// TIA Portal V18 export
// export: Created 2026-03-12T16:04:35.3703987Z, ExportSetting WithDefaults, DisplayName Totally Integrated Automation Portal, DisplayVersion V18 Update 5, DisplayName TIA Portal Openness, DisplayVersion V18 Update 5, DisplayName TIA Portal Version Control Interface, DisplayVersion V18, DisplayName SINAMICS Startdrive Advanced, DisplayVersion V18, DisplayName SINAMICS Startdrive G130, G150, S120, S150, SINAMICS MV, S210, DisplayVersion V18, DisplayName SINAMICS Startdrive G110M, G120, G120C, G120D, G120P, G115D, DisplayVersion V18, DisplayName STEP 7 Professional, DisplayVersion V18 Update 5, DisplayName STEP 7 Safety, DisplayVersion V18, DisplayName WinCC Professional, DisplayVersion V18 Update 5
FUNCTION_BLOCK "FB LIMITES_OPERACAO_SENSOR"   // FB25, LAD
{ S7_Optimized_Access := 'TRUE' }
VERSION : 0.1
// stored: AutoNumber true, IsIECCheckEnabled false, IsRetainMemResEnabled false, MemoryReserve 100, SetENOAutomatically false, UDAEnableTagReadback false
   VAR_INPUT
      STATUS_SENSOR : Real;
      COMANDO : Int;
      COMANDO_VALOR : Int;
      ENTRADA_VALOR_MUITO_BAIXO : Real;
      ENTRADA_VALOR_BAIXO : Real;
      ENTRADA_VALOR_ALTO : Real;
      ENTRADA_VALOR_MUITO_ALTO : Real;
      COMANDO_MANUTENCAO : Bool;
      SEM_SINAL_4mA : Bool;
   END_VAR
   VAR_OUTPUT
      SAIDA_LEITURA_MUITO_BAIXA : Bool;
      SAIDA_LEITURA_BAIXO : Bool;
      SAIDA_LEITURA_ALTO : Bool;
      SAIDA_LEITURA_MUITO_ALTO : Bool;
   END_VAR
   VAR_IN_OUT
      VALOR_MUITO_BAIXO : Real;
      VALOR_BAIXO : Real;
      VALOR_ALTO : Real;
      VALOR_MUITO_ALTO : Real;
   END_VAR
   VAR
      TON_1 { ExternalAccessible := 'False'; ExternalVisible := 'False'; ExternalWritable := 'False'} : IEC_TIMER;
      TON_2 { ExternalAccessible := 'False'; ExternalVisible := 'False'; ExternalWritable := 'False'} : IEC_TIMER;
      TON_3 { ExternalAccessible := 'False'; ExternalVisible := 'False'; ExternalWritable := 'False'} : IEC_TIMER;
      TON_4 { ExternalAccessible := 'False'; ExternalVisible := 'False'; ExternalWritable := 'False'} : IEC_TIMER;
   END_VAR
   VAR_TEMP   // added for the SCL form of the ladder/FBD networks
      _w1 : Bool;
   END_VAR
BEGIN

REGION Network 1: Carrega valor de referencia
   // Network responsável por carregar os valores de referência (setpoints)
   //  para os limites do Medidor, com base em um comando de seleção de valor.
   //  O valor em '#COMANDO' determina qual conjunto de limites será ativo.
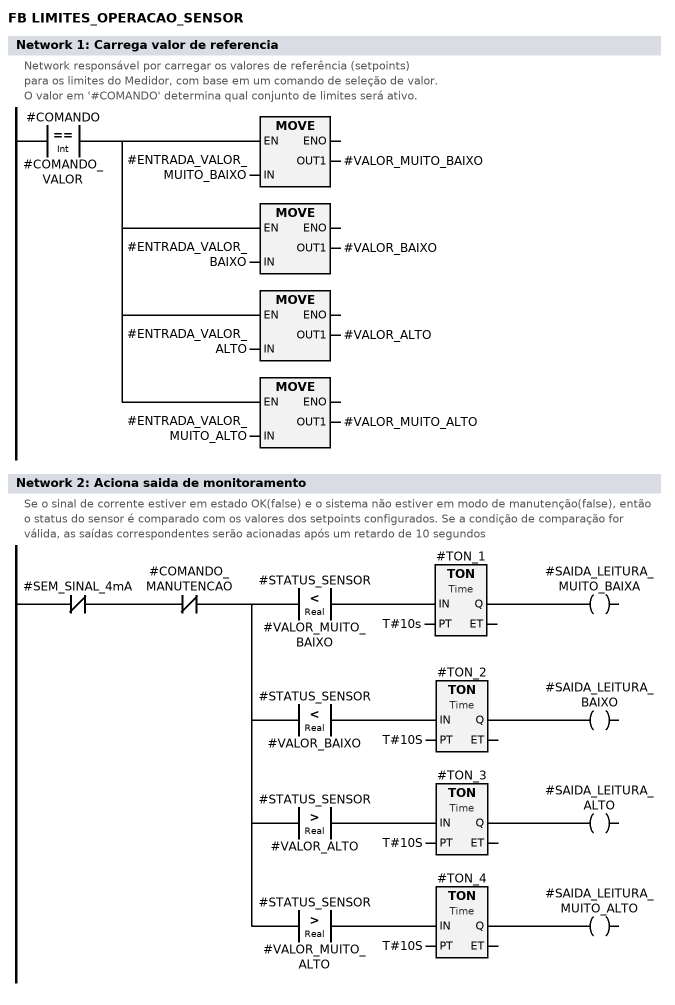
   RUNG wire#powerrail
      { S7_Templates := "SrcType := Int" } EQ_Contact(in1 := #COMANDO, in2 := #COMANDO_VALOR)
      wire#w1
      Move(in := #ENTRADA_VALOR_MUITO_BAIXO, out1 => #VALOR_MUITO_BAIXO)
   END_RUNG
   RUNG wire#w1
      Move(in := #ENTRADA_VALOR_BAIXO, out1 => #VALOR_BAIXO)
   END_RUNG
   RUNG wire#w1
      Move(in := #ENTRADA_VALOR_ALTO, out1 => #VALOR_ALTO)
   END_RUNG
   RUNG wire#w1
      Move(in := #ENTRADA_VALOR_MUITO_ALTO, out1 => #VALOR_MUITO_ALTO)
   END_RUNG
   // the same network as SCL:
   IF #COMANDO = #COMANDO_VALOR THEN
       #VALOR_MUITO_BAIXO := #ENTRADA_VALOR_MUITO_BAIXO;
       #VALOR_BAIXO := #ENTRADA_VALOR_BAIXO;
       #VALOR_ALTO := #ENTRADA_VALOR_ALTO;
       #VALOR_MUITO_ALTO := #ENTRADA_VALOR_MUITO_ALTO;
   END_IF;
END_REGION

REGION Network 2: Aciona saida de monitoramento
   // Se o sinal de corrente estiver em estado OK(false) e o sistema não estiver em modo de manutenção(false), então o status do sensor é comparado com os valores dos setpoints configurados. Se a condição de comparação for válida, as saídas correspondentes serão acionadas após um retardo de 10 segundos
   RUNG wire#powerrail
      I_Contact( #SEM_SINAL_4mA )
      I_Contact( #COMANDO_MANUTENCAO )
      wire#w1
      { S7_Templates := "SrcType := Real" } LT_Contact(in1 := #STATUS_SENSOR, in2 := #VALOR_MUITO_BAIXO)
      { S7_Templates := "time_type := Time" } #TON_1.TON(pt := T#10s, et =>)
      Coil( #SAIDA_LEITURA_MUITO_BAIXA )
   END_RUNG
   RUNG wire#w1
      { S7_Templates := "SrcType := Real" } LT_Contact(in1 := #STATUS_SENSOR, in2 := #VALOR_BAIXO)
      { S7_Templates := "time_type := Time" } #TON_2.TON(pt := T#10S, et =>)
      Coil( #SAIDA_LEITURA_BAIXO )
   END_RUNG
   RUNG wire#w1
      { S7_Templates := "SrcType := Real" } GT_Contact(in1 := #STATUS_SENSOR, in2 := #VALOR_ALTO)
      { S7_Templates := "time_type := Time" } #TON_3.TON(pt := T#10S, et =>)
      Coil( #SAIDA_LEITURA_ALTO )
   END_RUNG
   RUNG wire#w1
      { S7_Templates := "SrcType := Real" } GT_Contact(in1 := #STATUS_SENSOR, in2 := #VALOR_MUITO_ALTO)
      { S7_Templates := "time_type := Time" } #TON_4.TON(pt := T#10S, et =>)
      Coil( #SAIDA_LEITURA_MUITO_ALTO )
   END_RUNG
   // the same network as SCL:
   #_w1 := NOT #SEM_SINAL_4mA AND NOT #COMANDO_MANUTENCAO;
   #TON_1.TON(IN := #_w1 AND (#STATUS_SENSOR < #VALOR_MUITO_BAIXO), PT := T#10s);
   #SAIDA_LEITURA_MUITO_BAIXA := #TON_1.Q;
   #TON_2.TON(IN := #_w1 AND (#STATUS_SENSOR < #VALOR_BAIXO), PT := T#10S);
   #SAIDA_LEITURA_BAIXO := #TON_2.Q;
   #TON_3.TON(IN := #_w1 AND (#STATUS_SENSOR > #VALOR_ALTO), PT := T#10S);
   #SAIDA_LEITURA_ALTO := #TON_3.Q;
   #TON_4.TON(IN := #_w1 AND (#STATUS_SENSOR > #VALOR_MUITO_ALTO), PT := T#10S);
   #SAIDA_LEITURA_MUITO_ALTO := #TON_4.Q;
END_REGION
END_FUNCTION_BLOCK
